(* Logix 5000 project; controller CarbonScout_MK6 vendor 1 type 14 code 154 rev 32.11; software revision 32.00; part 15 of 17 *)
(* tags used below, declared in another part *)
   CNT : DINT;
   DN_Cal : BOOL;   // Calculation Done Bit to proceed next step
   LocalSampleTank : DINT;
   LOnlineNumber : DINT;
   ONS : BOOL[32];
   SampleIndexNum : DINT;
   storage : BOOL;
   XRF_ReadyTimer : TIMER;
   CS_Alarms : P_Alarm[80];
   CS_DINTParams : DINT[100];
   CS_REALParams : REAL[80];   // CS REAL Parameters
   CS_Result : CS_Results;   // Sample Result Live Async
   CS_ResultsSync : CS_Results;
   CS_SampleSeq : DINT[129];
   CS_Seq : GEK_Sequence;
   CS_Tank : CS_TankParams[20];
   CS_Timer : TIMER[80];
   CS_Timer2 : TIMER[20];
   CS_XRF : XRF;
   CS_XRF_Elements : LinearModelXRF;   // Linear model 0 is inital factory model and 1 is trimming model
   CS_XRF_RawModel : REAL[4];
   N51 : DINT[5];   // From Client
   Oneshot : DINT;
   Oneshot2 : DINT;
   Oneshot3 : DINT;
   Reg_Model : REAL[4];   // Calculated model output and site model
   TankPointer : DINT;
   test : DINT;
   Valve_XV_15 : P_ValveSO;   // Bottme wash vavle
   Valve_XV_19 : P_ValveSO;   // Laser window
   Valve_XV_40 : P_ValveSO;   // XRF power on valve
   XRF_RAWDINT : DINT[100];
(* SeqProgram, continued *)

ROUTINE TankSelection   (* ladder *)
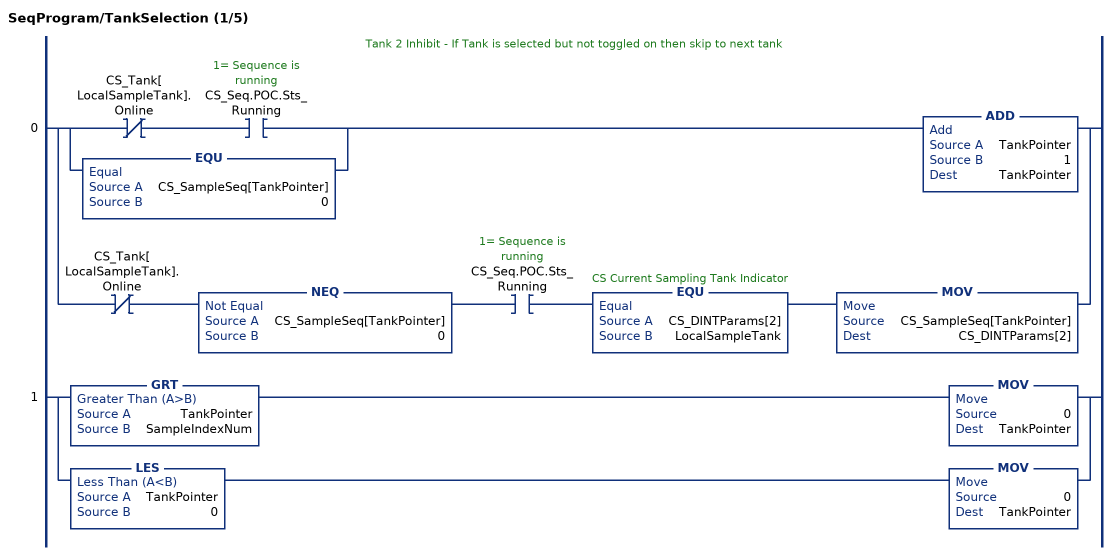
   // Tank 2 Inhibit - If Tank is selected but not toggled on then skip to next tank
   0: [[XIO(CS_Tank[LocalSampleTank].Online) XIC(CS_Seq.POC.Sts_Running) ,EQU(CS_SampleSeq[TankPointer],0) ] ADD(TankPointer,1,TankPointer) ,XIO(CS_Tank[LocalSampleTank].Online) NEQ(CS_SampleSeq[TankPointer],0) XIC(CS_Seq.POC.Sts_Running) EQU(CS_DINTParams[2],LocalSampleTank) MOV(CS_SampleSeq[TankPointer],CS_DINTParams[2]) ];
   1: [GRT(TankPointer,SampleIndexNum) MOV(0,TankPointer) ,LES(TankPointer,0) MOV(0,TankPointer) ];
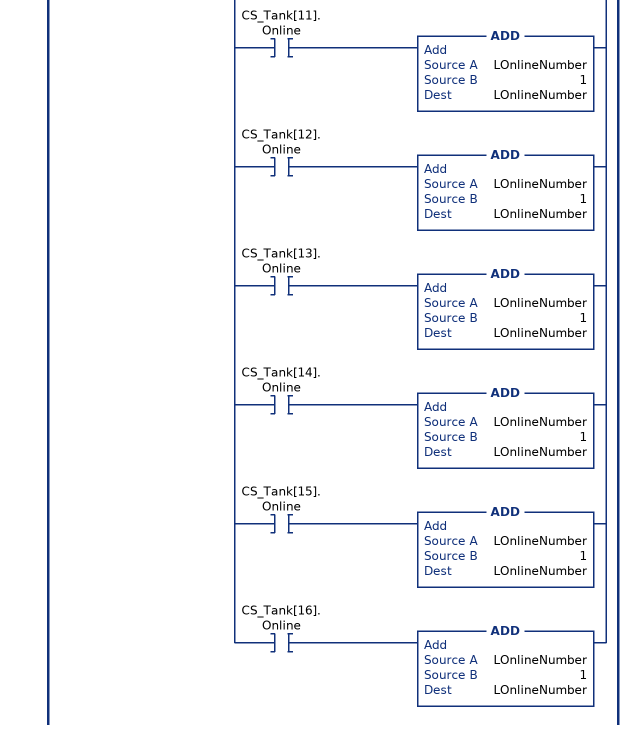
   2: CLR(LOnlineNumber)[XIC(CS_Tank[1].Online) ADD(LOnlineNumber,1,LOnlineNumber) ,XIC(CS_Tank[2].Online) ADD(LOnlineNumber,1,LOnlineNumber) ,XIC(CS_Tank[3].Online) ADD(LOnlineNumber,1,LOnlineNumber) ,XIC(CS_Tank[4].Online) ADD(LOnlineNumber,1,LOnlineNumber) ,XIC(CS_Tank[5].Online) ADD(LOnlineNumber,1,LOnlineNumber) ,XIC(CS_Tank[6].Online) ADD(LOnlineNumber,1,LOnlineNumber) ,XIC(CS_Tank[7].Online) ADD(LOnlineNumber,1,LOnlineNumber) ,XIC(CS_Tank[8].Online) ADD(LOnlineNumber,1,LOnlineNumber) ,XIC(CS_Tank[9].Online) ADD(LOnlineNumber,1,LOnlineNumber) ,XIC(CS_Tank[10].Online) ADD(LOnlineNumber,1,LOnlineNumber) ,XIC(CS_Tank[11].Online) ADD(LOnlineNumber,1,LOnlineNumber) ,XIC(CS_Tank[12].Online) ADD(LOnlineNumber,1,LOnlineNumber) ,XIC(CS_Tank[13].Online) ADD(LOnlineNumber,1,LOnlineNumber) ,XIC(CS_Tank[14].Online) ADD(LOnlineNumber,1,LOnlineNumber) ,XIC(CS_Tank[15].Online) ADD(LOnlineNumber,1,LOnlineNumber) ,XIC(CS_Tank[16].Online) ADD(LOnlineNumber,1,LOnlineNumber) ];
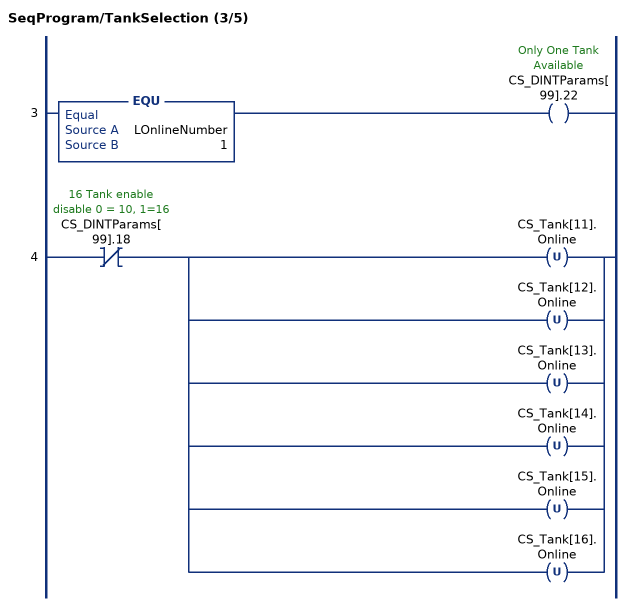
   3: EQU(LOnlineNumber,1)OTE(CS_DINTParams[99].22);
   4: XIO(CS_DINTParams[99].18)[OTU(CS_Tank[11].Online) ,OTU(CS_Tank[12].Online) ,OTU(CS_Tank[13].Online) ,OTU(CS_Tank[14].Online) ,OTU(CS_Tank[15].Online) ,OTU(CS_Tank[16].Online) ];
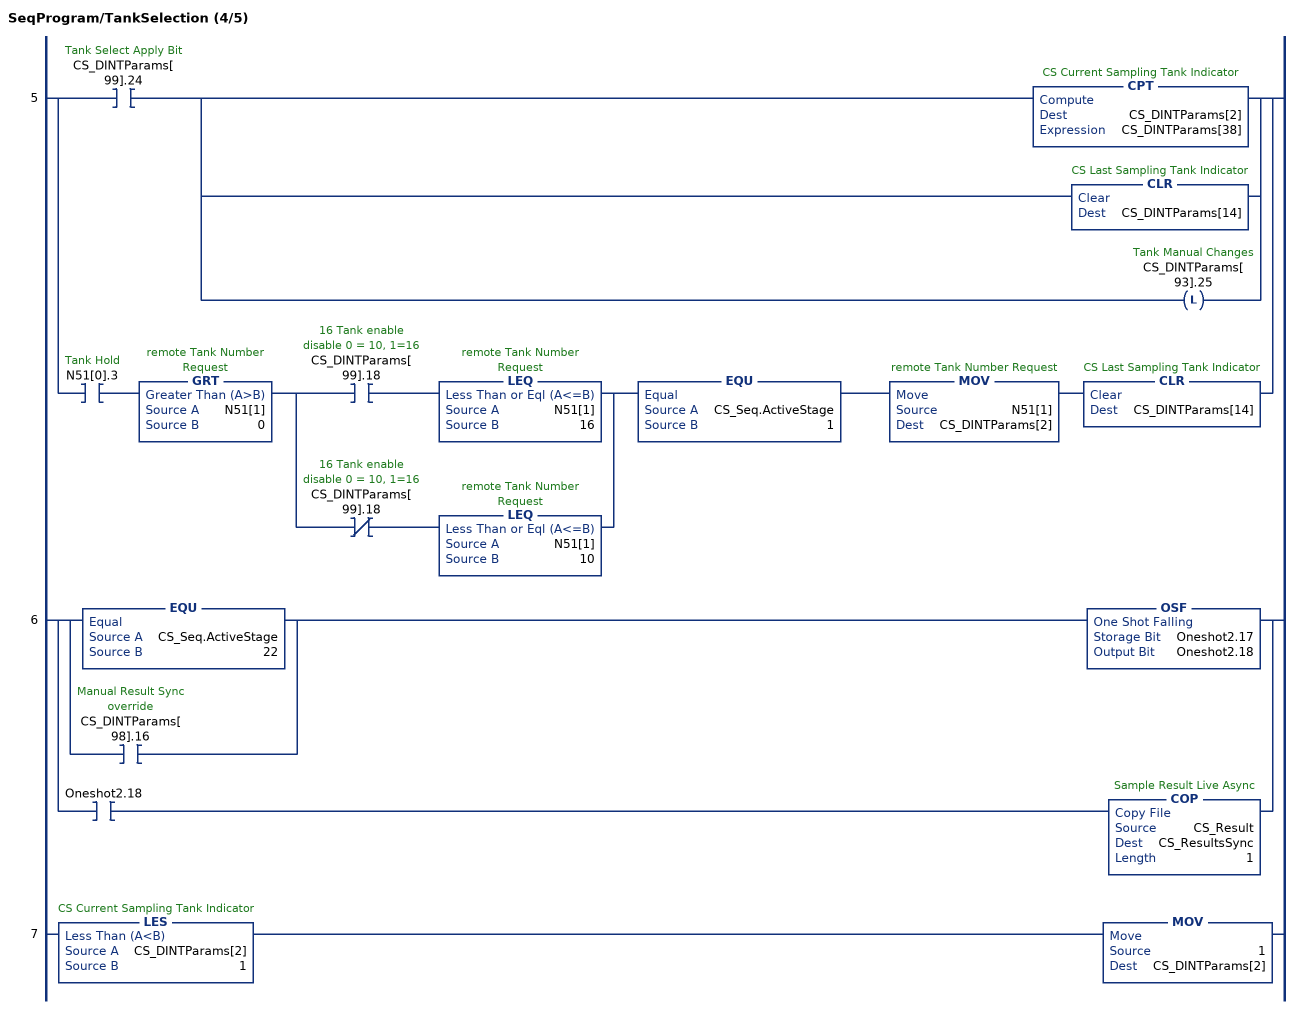
   5: [XIC(CS_DINTParams[99].24) [[CPT(CS_DINTParams[2],CS_DINTParams[38]) ,CLR(CS_DINTParams[14]) ] ,OTL(CS_DINTParams[93].25) ] ,XIC(N51[0].3) GRT(N51[1],0) [XIC(CS_DINTParams[99].18) LEQ(N51[1],16) ,XIO(CS_DINTParams[99].18) LEQ(N51[1],10) ] EQU(CS_Seq.ActiveStage,1) MOV(N51[1],CS_DINTParams[2]) CLR(CS_DINTParams[14]) ];
   6: [[EQU(CS_Seq.ActiveStage,22) ,XIC(CS_DINTParams[98].16) ] OSF(Oneshot2.17,Oneshot2.18) ,XIC(Oneshot2.18) COP(CS_Result,CS_ResultsSync,1) ];
   7: LES(CS_DINTParams[2],1)MOV(1,CS_DINTParams[2]);
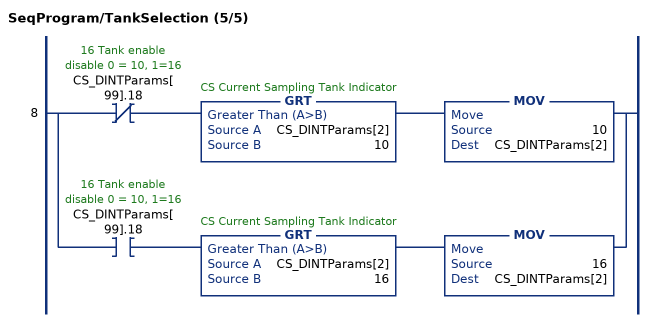
   8: [XIO(CS_DINTParams[99].18) GRT(CS_DINTParams[2],10) MOV(10,CS_DINTParams[2]) ,XIC(CS_DINTParams[99].18) GRT(CS_DINTParams[2],16) MOV(16,CS_DINTParams[2]) ];
END_ROUTINE

ROUTINE XRF   (* ladder *)
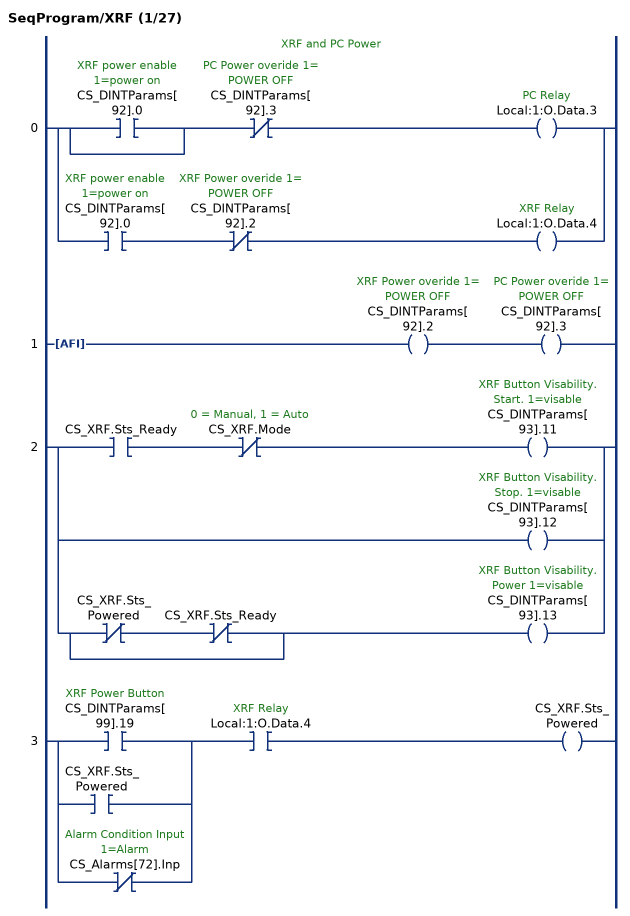
   // XRF and PC Power
   0: [[XIC(CS_DINTParams[92].0) ,] XIO(CS_DINTParams[92].3) OTE(Local:1:O.Data.3) ,XIC(CS_DINTParams[92].0) XIO(CS_DINTParams[92].2) OTE(Local:1:O.Data.4) ];
   1: AFI()OTE(CS_DINTParams[92].2)OTE(CS_DINTParams[92].3);
   2: [XIC(CS_XRF.Sts_Ready) XIO(CS_XRF.Mode) OTE(CS_DINTParams[93].11) ,OTE(CS_DINTParams[93].12) ,[XIO(CS_XRF.Sts_Powered) XIO(CS_XRF.Sts_Ready) ,] OTE(CS_DINTParams[93].13) ];
   3: [XIC(CS_DINTParams[99].19) ,XIC(CS_XRF.Sts_Powered) ,XIO(CS_Alarms[72].Inp) ]XIC(Local:1:O.Data.4)OTE(CS_XRF.Sts_Powered);
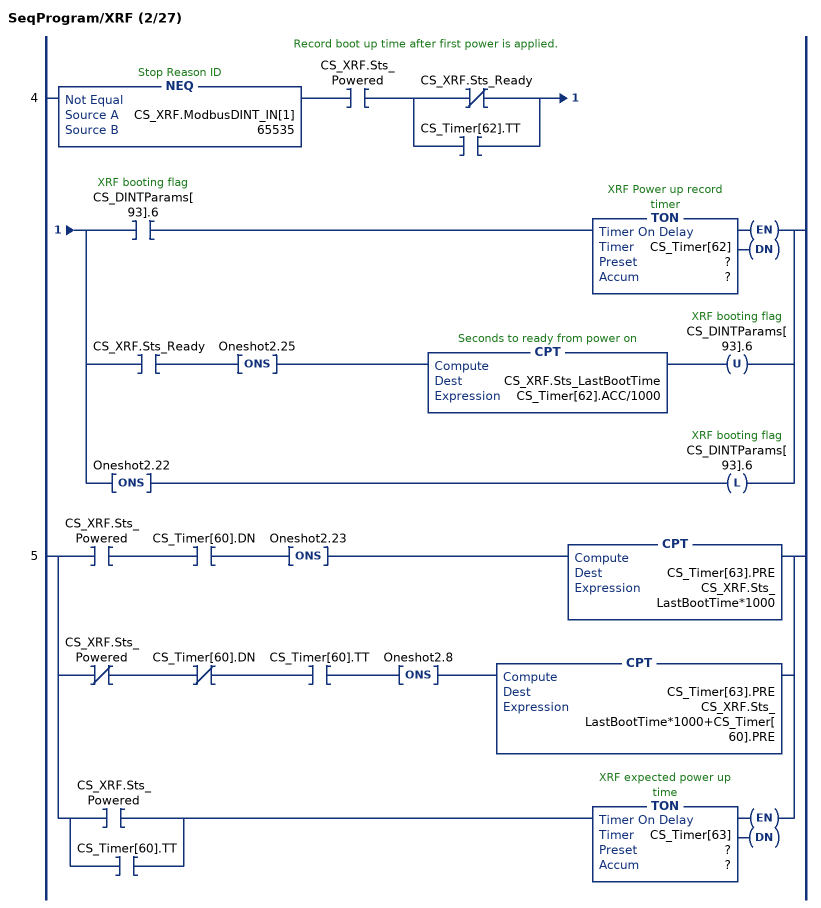
   // Record boot up time after first power is applied.
   4: NEQ(CS_XRF.ModbusDINT_IN[1],65535)XIC(CS_XRF.Sts_Powered)[XIO(CS_XRF.Sts_Ready) ,XIC(CS_Timer[62].TT) ][XIC(CS_DINTParams[93].6) TON(CS_Timer[62],?,?) ,XIC(CS_XRF.Sts_Ready) ONS(Oneshot2.25) CPT(CS_XRF.Sts_LastBootTime,CS_Timer[62].ACC/1000) OTU(CS_DINTParams[93].6) ,ONS(Oneshot2.22) OTL(CS_DINTParams[93].6) ];
   5: [XIC(CS_XRF.Sts_Powered) XIC(CS_Timer[60].DN) ONS(Oneshot2.23) CPT(CS_Timer[63].PRE,CS_XRF.Sts_LastBootTime*1000) ,XIO(CS_XRF.Sts_Powered) XIO(CS_Timer[60].DN) XIC(CS_Timer[60].TT) ONS(Oneshot2.8) CPT(CS_Timer[63].PRE,CS_XRF.Sts_LastBootTime*1000+CS_Timer[60].PRE) ,[XIC(CS_XRF.Sts_Powered) ,XIC(CS_Timer[60].TT) ] TON(CS_Timer[63],?,?) ];
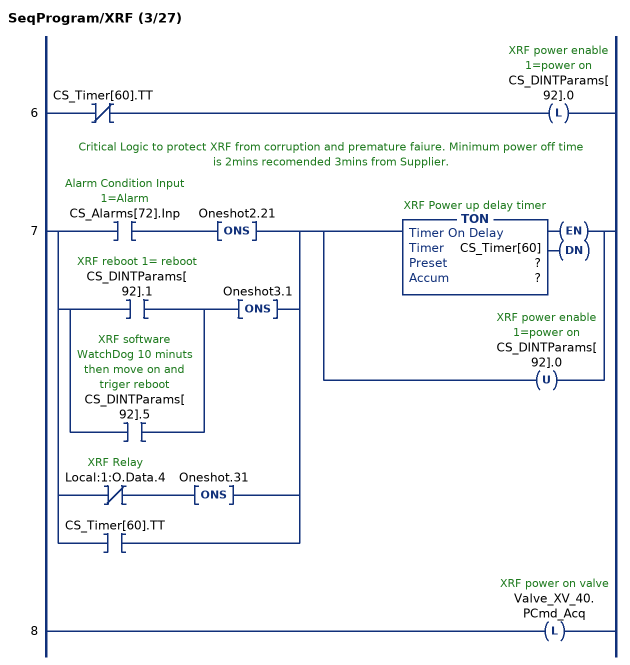
   6: XIO(CS_Timer[60].TT)OTL(CS_DINTParams[92].0);
   // Critical Logic to protect XRF from corruption and premature faiure. Minimum power off time is 2mins recomended 3mins from Supplier.
   7: [XIC(CS_Alarms[72].Inp) ONS(Oneshot2.21) ,[XIC(CS_DINTParams[92].1) ,XIC(CS_DINTParams[92].5) ] ONS(Oneshot3.1) ,XIO(Local:1:O.Data.4) ONS(Oneshot.31) ,XIC(CS_Timer[60].TT) ][TON(CS_Timer[60],?,?) ,OTU(CS_DINTParams[92].0) ];
   8: OTL(Valve_XV_40.PCmd_Acq);
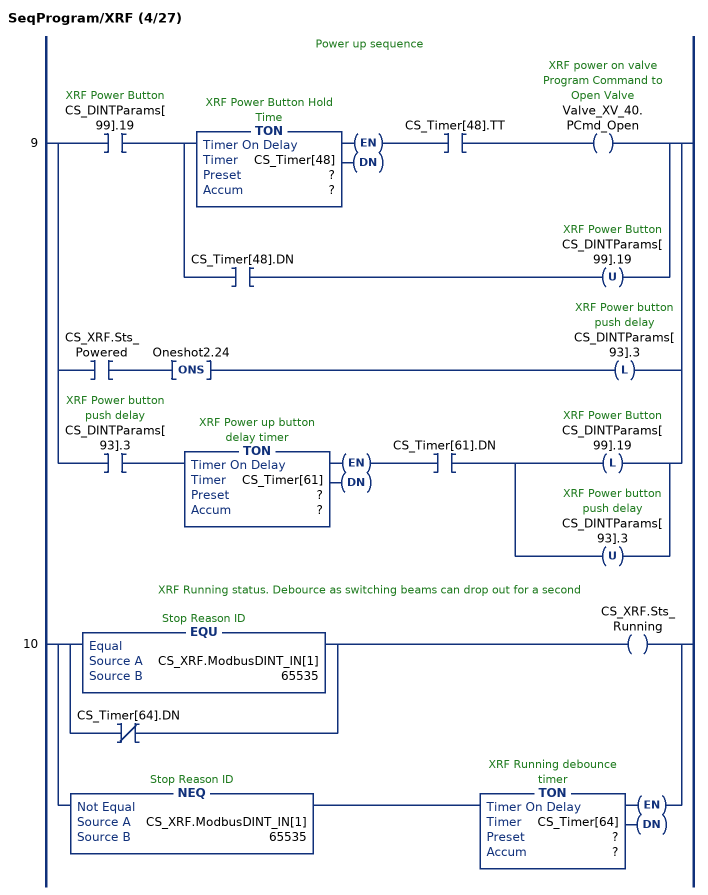
   // Power up sequence
   9: [XIC(CS_DINTParams[99].19) [TON(CS_Timer[48],?,?) XIC(CS_Timer[48].TT) OTE(Valve_XV_40.PCmd_Open) ,XIC(CS_Timer[48].DN) OTU(CS_DINTParams[99].19) ] ,XIC(CS_XRF.Sts_Powered) ONS(Oneshot2.24) OTL(CS_DINTParams[93].3) ,XIC(CS_DINTParams[93].3) TON(CS_Timer[61],?,?) XIC(CS_Timer[61].DN) [OTL(CS_DINTParams[99].19) ,OTU(CS_DINTParams[93].3) ] ];
   // XRF Running status. Debource as switching beams can drop out for a second
   10: [[EQU(CS_XRF.ModbusDINT_IN[1],65535) ,XIO(CS_Timer[64].DN) ] OTE(CS_XRF.Sts_Running) ,NEQ(CS_XRF.ModbusDINT_IN[1],65535) TON(CS_Timer[64],?,?) ];
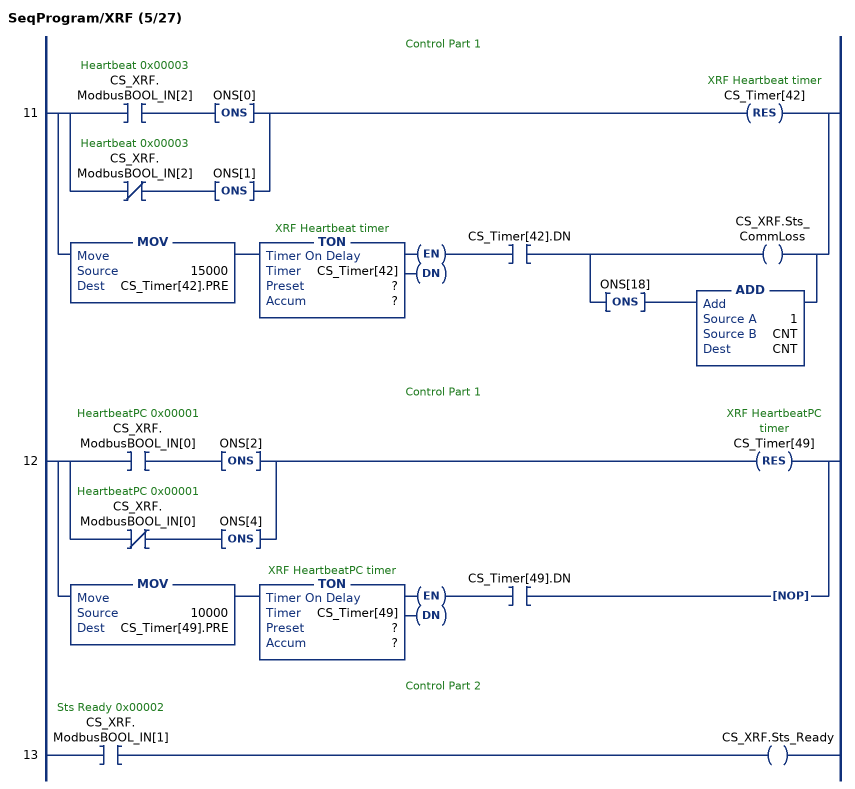
   // Control Part 1
   11: [[XIC(CS_XRF.ModbusBOOL_IN[2]) ONS(ONS[0]) ,XIO(CS_XRF.ModbusBOOL_IN[2]) ONS(ONS[1]) ] RES(CS_Timer[42]) ,MOV(15000,CS_Timer[42].PRE) TON(CS_Timer[42],?,?) XIC(CS_Timer[42].DN) [OTE(CS_XRF.Sts_CommLoss) ,ONS(ONS[18]) ADD(1,CNT,CNT) ] ];
   // Control Part 1
   12: [[XIC(CS_XRF.ModbusBOOL_IN[0]) ONS(ONS[2]) ,XIO(CS_XRF.ModbusBOOL_IN[0]) ONS(ONS[4]) ] RES(CS_Timer[49]) ,MOV(10000,CS_Timer[49].PRE) TON(CS_Timer[49],?,?) XIC(CS_Timer[49].DN) NOP() ];
   // Control Part 2
   13: XIC(CS_XRF.ModbusBOOL_IN[1])OTE(CS_XRF.Sts_Ready);
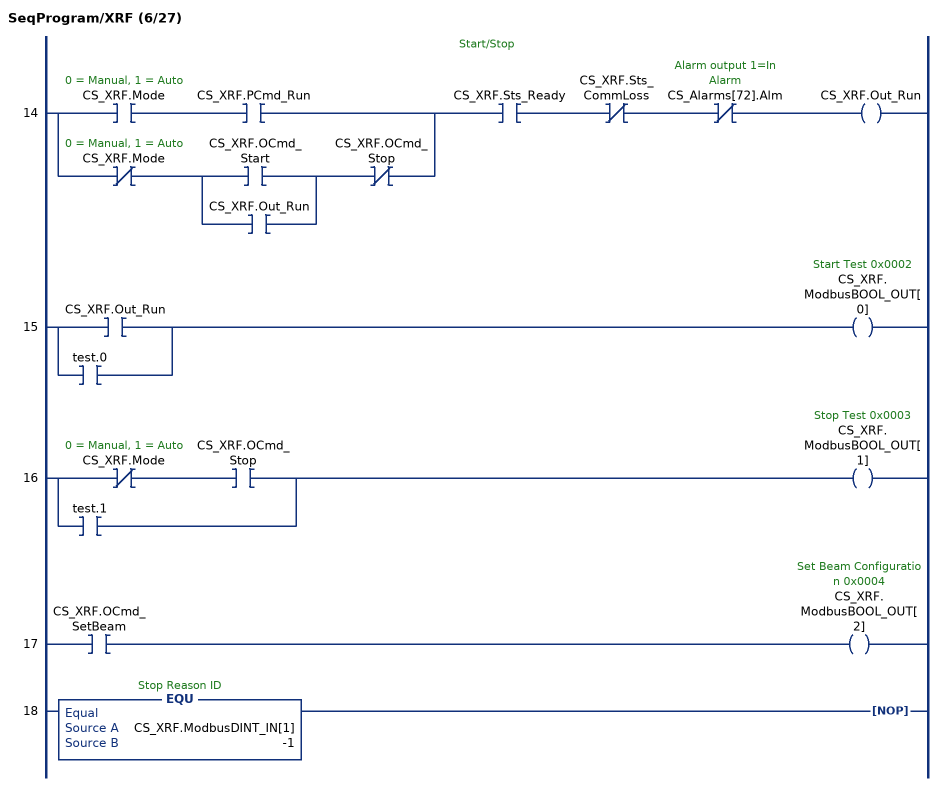
   // Start/Stop
   14: [XIC(CS_XRF.Mode) XIC(CS_XRF.PCmd_Run) ,XIO(CS_XRF.Mode) [XIC(CS_XRF.OCmd_Start) ,XIC(CS_XRF.Out_Run) ] XIO(CS_XRF.OCmd_Stop) ]XIC(CS_XRF.Sts_Ready)XIO(CS_XRF.Sts_CommLoss)XIO(CS_Alarms[72].Alm)OTE(CS_XRF.Out_Run);
   15: [XIC(CS_XRF.Out_Run) ,XIC(test.0) ]OTE(CS_XRF.ModbusBOOL_OUT[0]);
   16: [XIO(CS_XRF.Mode) XIC(CS_XRF.OCmd_Stop) ,XIC(test.1) ]OTE(CS_XRF.ModbusBOOL_OUT[1]);
   17: XIC(CS_XRF.OCmd_SetBeam)OTE(CS_XRF.ModbusBOOL_OUT[2]);
   18: EQU(CS_XRF.ModbusDINT_IN[1],-1)NOP();
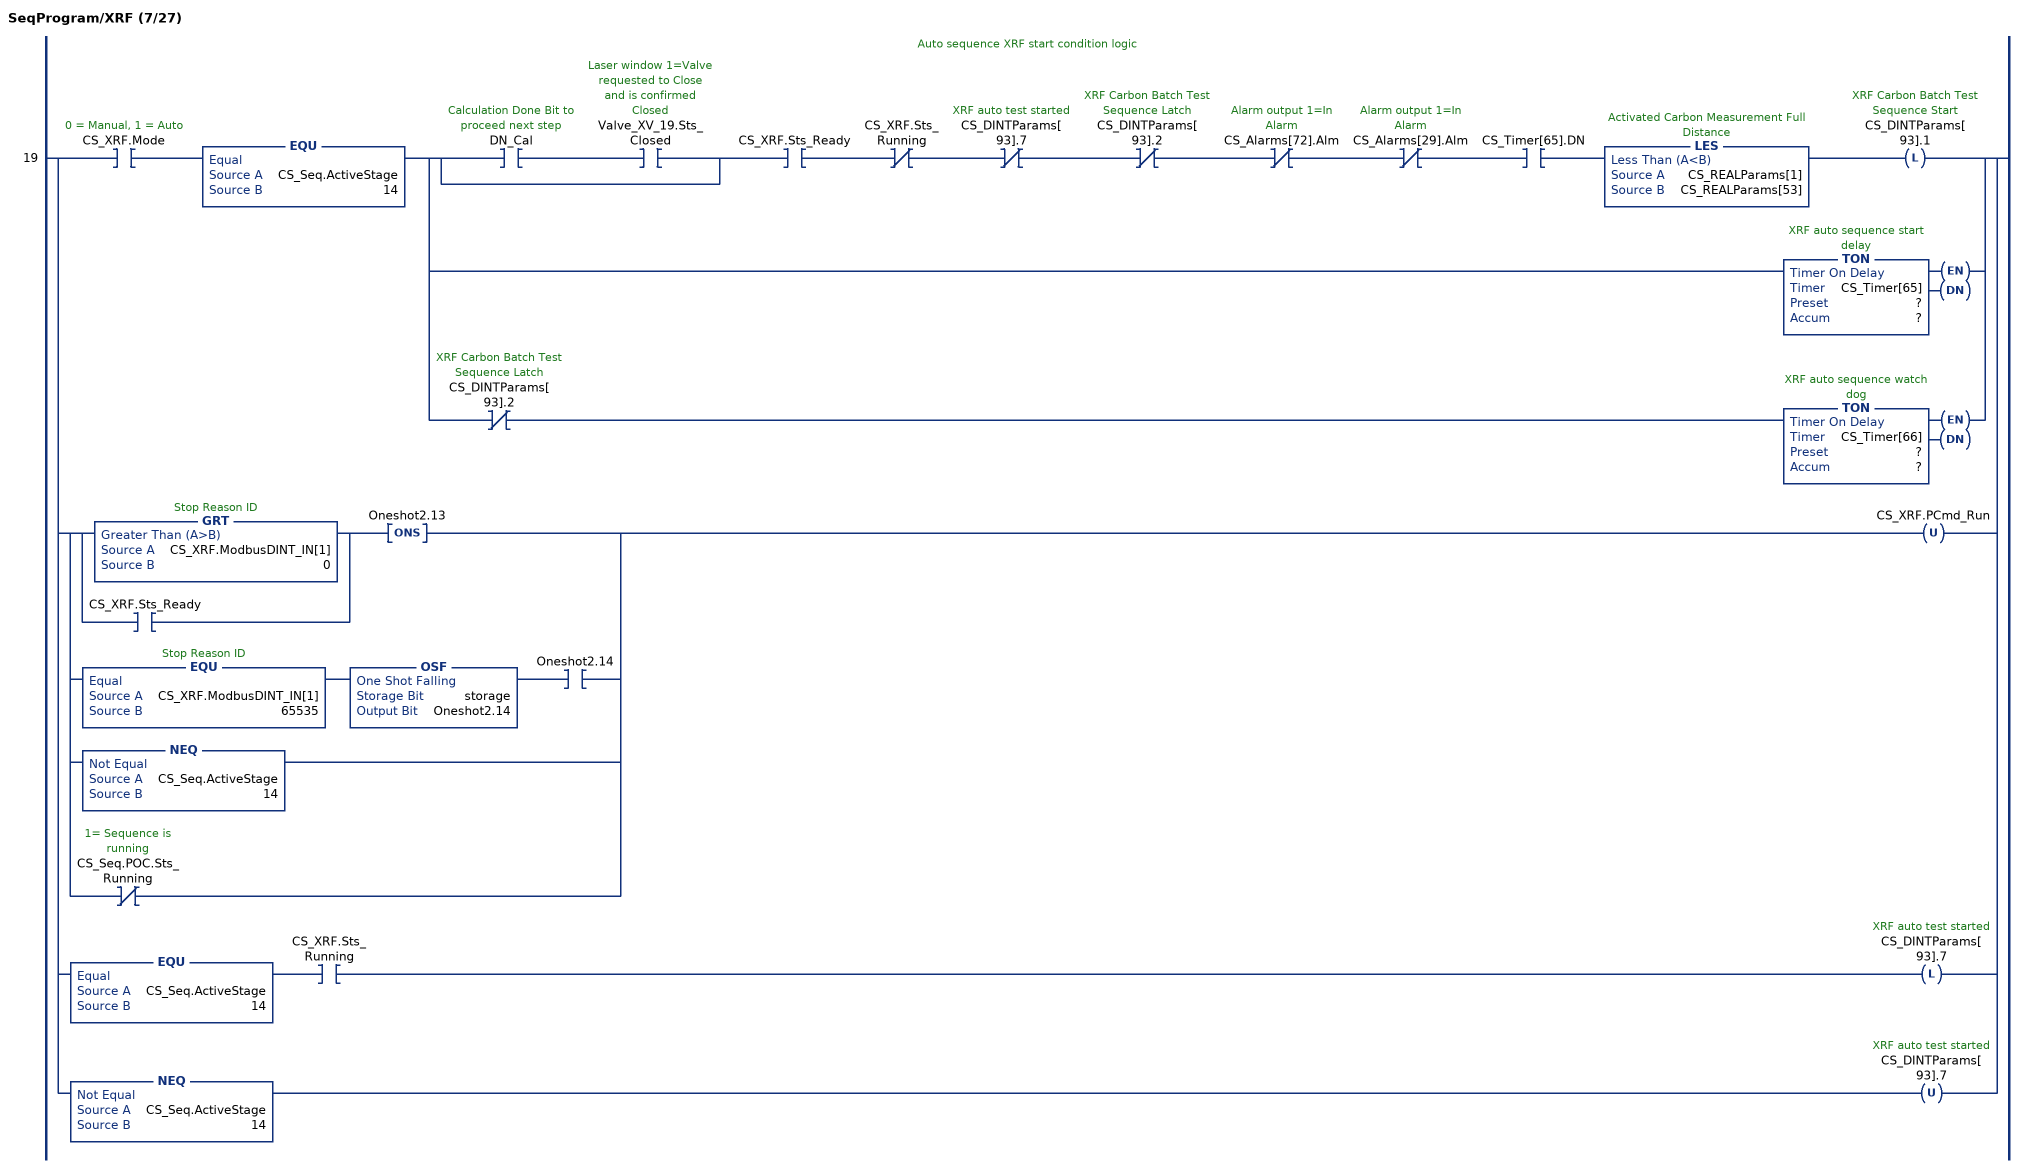
   // Auto sequence XRF start condition logic
   19: [XIC(CS_XRF.Mode) EQU(CS_Seq.ActiveStage,14) [[XIC(DN_Cal) XIC(Valve_XV_19.Sts_Closed) ,] XIC(CS_XRF.Sts_Ready) XIO(CS_XRF.Sts_Running) XIO(CS_DINTParams[93].7) XIO(CS_DINTParams[93].2) XIO(CS_Alarms[72].Alm) XIO(CS_Alarms[29].Alm) XIC(CS_Timer[65].DN) LES(CS_REALParams[1],CS_REALParams[53]) OTL(CS_DINTParams[93].1) ,[TON(CS_Timer[65],?,?) ,XIO(CS_DINTParams[93].2) TON(CS_Timer[66],?,?) ] ] ,[[GRT(CS_XRF.ModbusDINT_IN[1],0) ,XIC(CS_XRF.Sts_Ready) ] ONS(Oneshot2.13) ,EQU(CS_XRF.ModbusDINT_IN[1],65535) OSF(storage,Oneshot2.14) XIC(Oneshot2.14) ,NEQ(CS_Seq.ActiveStage,14) ,XIO(CS_Seq.POC.Sts_Running) ] OTU(CS_XRF.PCmd_Run) ,EQU(CS_Seq.ActiveStage,14) XIC(CS_XRF.Sts_Running) OTL(CS_DINTParams[93].7) ,NEQ(CS_Seq.ActiveStage,14) OTU(CS_DINTParams[93].7) ];
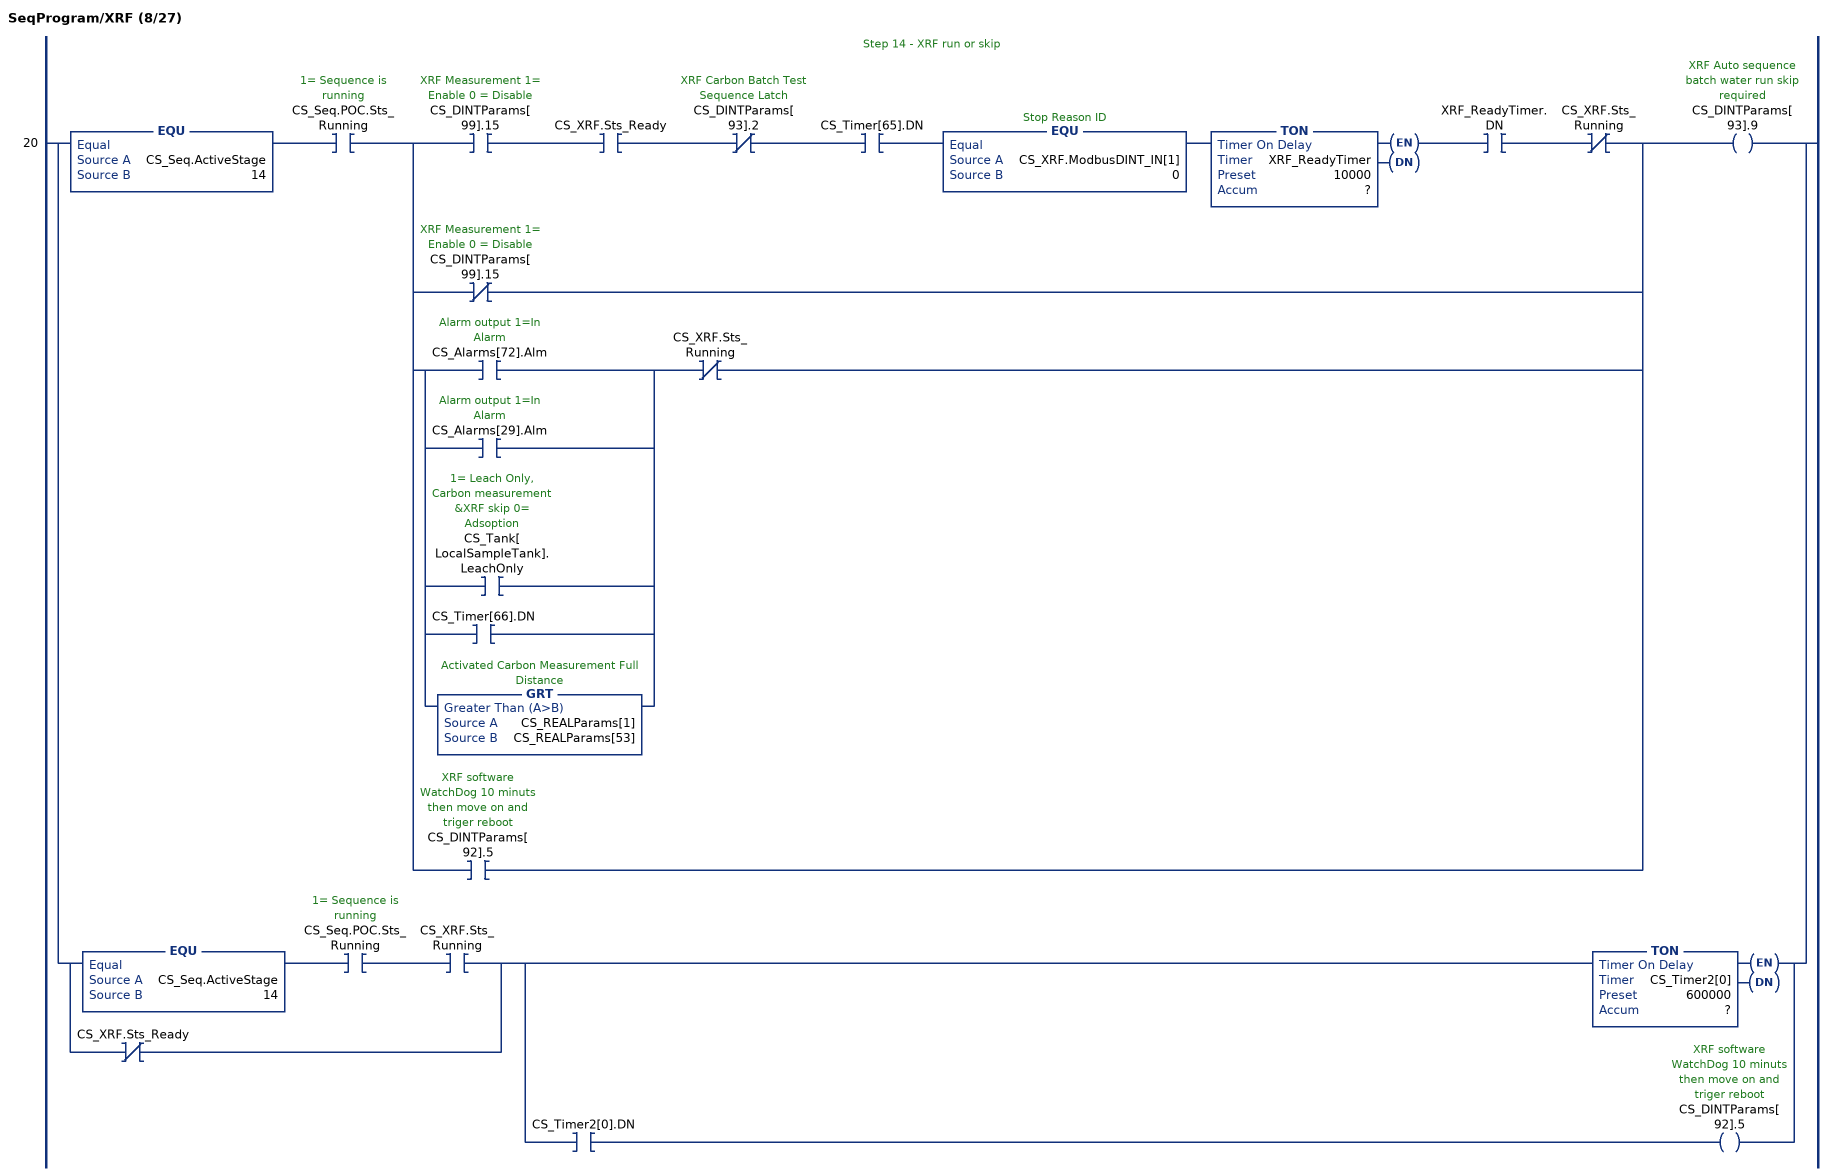
   // Step 14 - XRF run or skip
   20: [EQU(CS_Seq.ActiveStage,14) XIC(CS_Seq.POC.Sts_Running) [[XIC(CS_DINTParams[99].15) XIC(CS_XRF.Sts_Ready) XIO(CS_DINTParams[93].2) XIC(CS_Timer[65].DN) EQU(CS_XRF.ModbusDINT_IN[1],0) TON(XRF_ReadyTimer,?,?) XIC(XRF_ReadyTimer.DN) XIO(CS_XRF.Sts_Running) ,XIO(CS_DINTParams[99].15) ] ,[[XIC(CS_Alarms[72].Alm) ,XIC(CS_Alarms[29].Alm) ,XIC(CS_Tank[LocalSampleTank].LeachOnly) ,XIC(CS_Timer[66].DN) ,GRT(CS_REALParams[1],CS_REALParams[53]) ] XIO(CS_XRF.Sts_Running) ,XIC(CS_DINTParams[92].5) ] ] OTE(CS_DINTParams[93].9) ,[EQU(CS_Seq.ActiveStage,14) XIC(CS_Seq.POC.Sts_Running) XIC(CS_XRF.Sts_Running) ,XIO(CS_XRF.Sts_Ready) ] [TON(CS_Timer2[0],?,?) ,XIC(CS_Timer2[0].DN) OTE(CS_DINTParams[92].5) ] ];
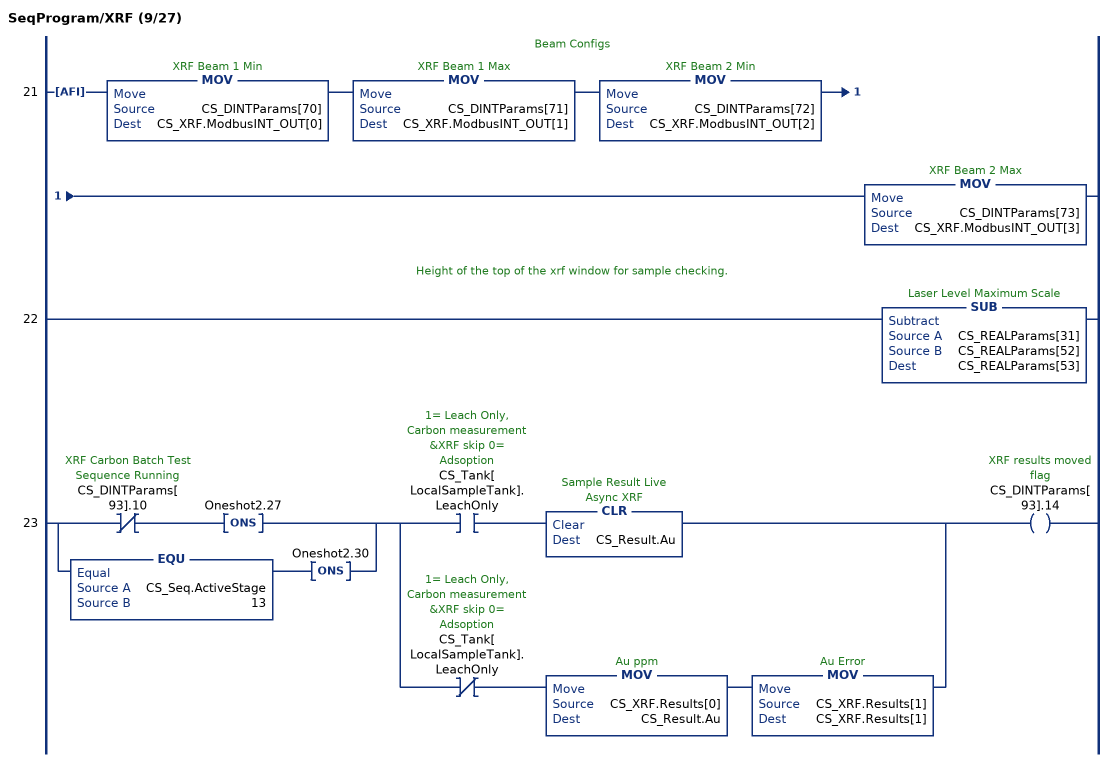
   // Beam Configs
   21: AFI()MOV(CS_DINTParams[70],CS_XRF.ModbusINT_OUT[0])MOV(CS_DINTParams[71],CS_XRF.ModbusINT_OUT[1])MOV(CS_DINTParams[72],CS_XRF.ModbusINT_OUT[2])MOV(CS_DINTParams[73],CS_XRF.ModbusINT_OUT[3]);
   // Height of the top of the xrf window for sample checking.
   22: SUB(CS_REALParams[31],CS_REALParams[52],CS_REALParams[53]);
   23: [XIO(CS_DINTParams[93].10) ONS(Oneshot2.27) ,EQU(CS_Seq.ActiveStage,13) ONS(Oneshot2.30) ][XIC(CS_Tank[LocalSampleTank].LeachOnly) CLR(CS_Result.Au) ,XIO(CS_Tank[LocalSampleTank].LeachOnly) MOV(CS_XRF.Results[0],CS_Result.Au) MOV(CS_XRF.Results[1],CS_XRF.Results[1]) ]OTE(CS_DINTParams[93].14);
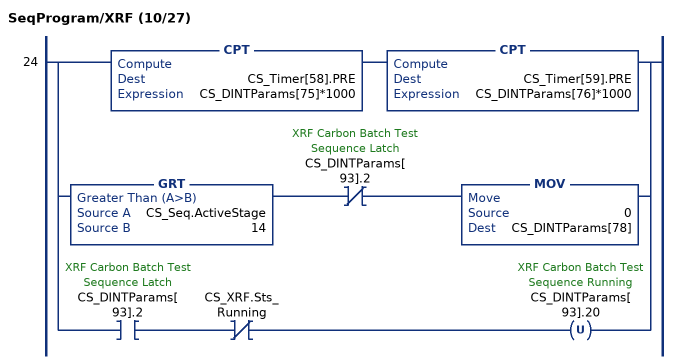
   24: [CPT(CS_Timer[58].PRE,CS_DINTParams[75]*1000) CPT(CS_Timer[59].PRE,CS_DINTParams[76]*1000) ,GRT(CS_Seq.ActiveStage,14) XIO(CS_DINTParams[93].2) MOV(0,CS_DINTParams[78]) ,XIC(CS_DINTParams[93].2) XIO(CS_XRF.Sts_Running) OTU(CS_DINTParams[93].20) ];
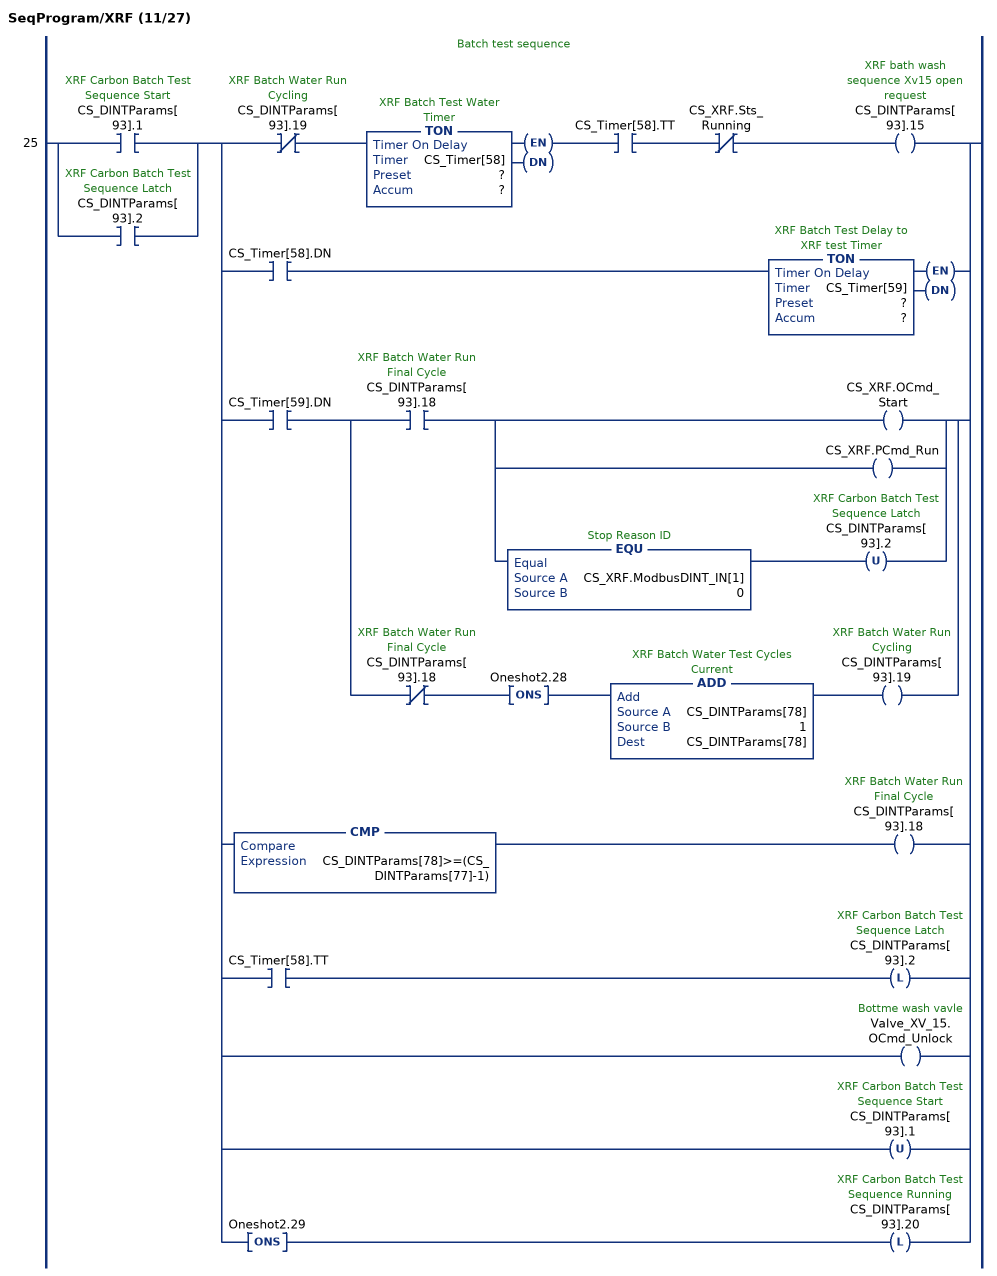
   // Batch test sequence
   25: [XIC(CS_DINTParams[93].1) ,XIC(CS_DINTParams[93].2) ][XIO(CS_DINTParams[93].19) TON(CS_Timer[58],?,?) XIC(CS_Timer[58].TT) XIO(CS_XRF.Sts_Running) OTE(CS_DINTParams[93].15) ,XIC(CS_Timer[58].DN) TON(CS_Timer[59],?,?) ,XIC(CS_Timer[59].DN) [XIC(CS_DINTParams[93].18) [[OTE(CS_XRF.OCmd_Start) ,OTE(CS_XRF.PCmd_Run) ] ,EQU(CS_XRF.ModbusDINT_IN[1],0) OTU(CS_DINTParams[93].2) ] ,XIO(CS_DINTParams[93].18) ONS(Oneshot2.28) ADD(CS_DINTParams[78],1,CS_DINTParams[78]) OTE(CS_DINTParams[93].19) ] ,CMP(CS_DINTParams[78]>=(CS_DINTParams[77]-1)) OTE(CS_DINTParams[93].18) ,XIC(CS_Timer[58].TT) OTL(CS_DINTParams[93].2) ,OTE(Valve_XV_15.OCmd_Unlock) ,OTU(CS_DINTParams[93].1) ,ONS(Oneshot2.29) OTL(CS_DINTParams[93].20) ];
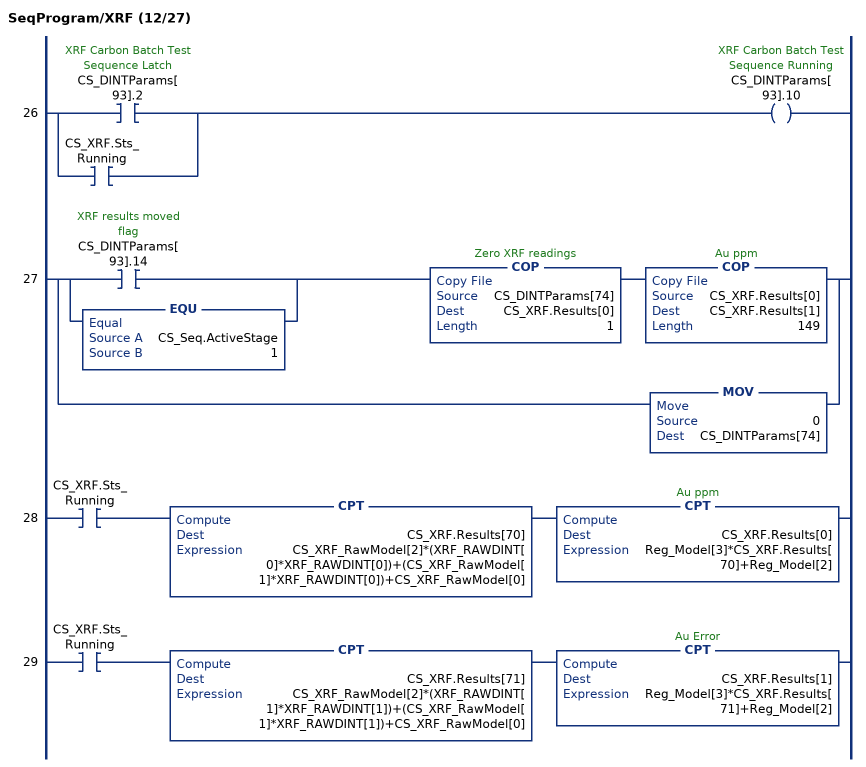
   26: [XIC(CS_DINTParams[93].2) ,XIC(CS_XRF.Sts_Running) ]OTE(CS_DINTParams[93].10);
   27: [[XIC(CS_DINTParams[93].14) ,EQU(CS_Seq.ActiveStage,1) ] COP(CS_DINTParams[74],CS_XRF.Results[0],1) COP(CS_XRF.Results[0],CS_XRF.Results[1],149) ,MOV(0,CS_DINTParams[74]) ];
   28: XIC(CS_XRF.Sts_Running)CPT(CS_XRF.Results[70],CS_XRF_RawModel[2]*(XRF_RAWDINT[0]*XRF_RAWDINT[0])+(CS_XRF_RawModel[1]*XRF_RAWDINT[0])+CS_XRF_RawModel[0])CPT(CS_XRF.Results[0],Reg_Model[3]*CS_XRF.Results[70]+Reg_Model[2]);
   29: XIC(CS_XRF.Sts_Running)CPT(CS_XRF.Results[71],CS_XRF_RawModel[2]*(XRF_RAWDINT[1]*XRF_RAWDINT[1])+(CS_XRF_RawModel[1]*XRF_RAWDINT[1])+CS_XRF_RawModel[0])CPT(CS_XRF.Results[1],Reg_Model[3]*CS_XRF.Results[71]+Reg_Model[2]);
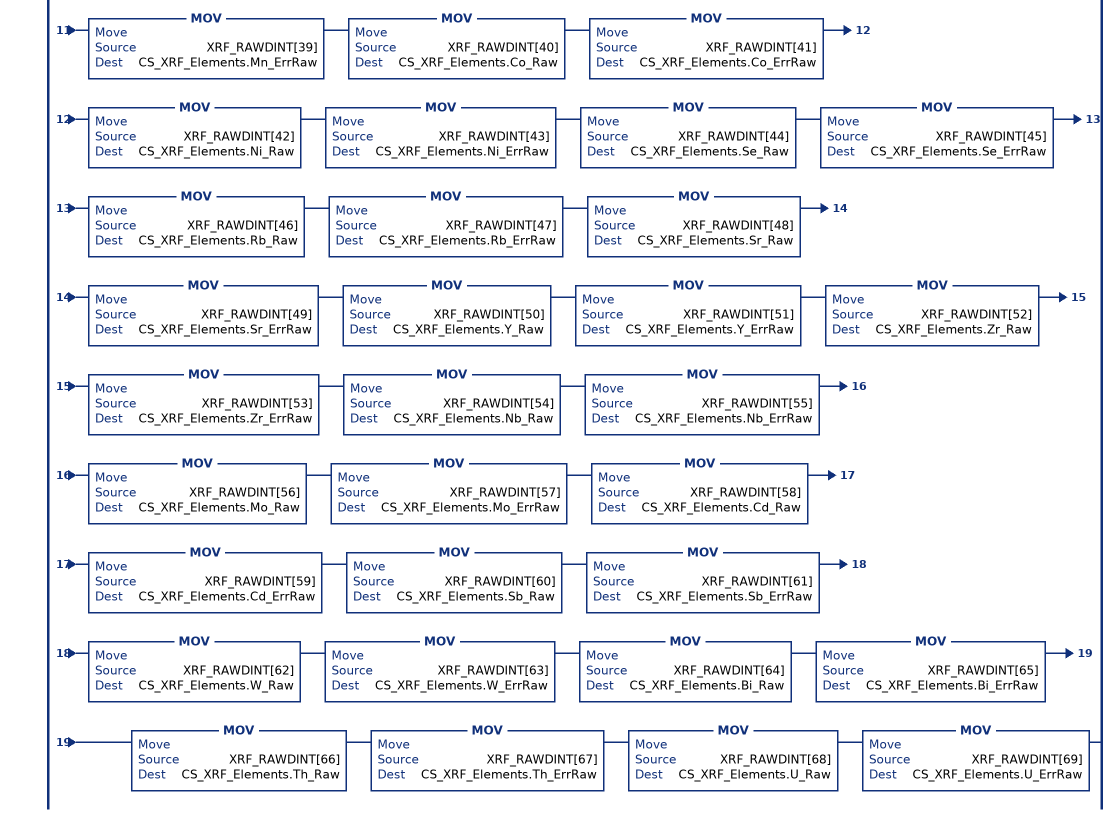
   30: MOV(XRF_RAWDINT[0],CS_XRF_Elements.Au_Raw)MOV(XRF_RAWDINT[1],CS_XRF_Elements.Au_ErrRaw)MOV(XRF_RAWDINT[2],CS_XRF_Elements.As_Raw)MOV(XRF_RAWDINT[3],CS_XRF_Elements.As_ErrRaw)MOV(XRF_RAWDINT[4],CS_XRF_Elements.Cu_Raw)MOV(XRF_RAWDINT[5],CS_XRF_Elements.Cu_ErrRaw)MOV(XRF_RAWDINT[6],CS_XRF_Elements.Fe_Raw)MOV(XRF_RAWDINT[7],CS_XRF_Elements.Fe_ErrRaw)MOV(XRF_RAWDINT[8],CS_XRF_Elements.Ag_Raw)MOV(XRF_RAWDINT[9],CS_XRF_Elements.Ag_ErrRaw)MOV(XRF_RAWDINT[10],CS_XRF_Elements.Hg_Raw)MOV(XRF_RAWDINT[11],CS_XRF_Elements.Hg_ErrRaw)MOV(XRF_RAWDINT[14],CS_XRF_Elements.Zn_Raw)MOV(XRF_RAWDINT[15],CS_XRF_Elements.Zn_ErrRaw)MOV(XRF_RAWDINT[16],CS_XRF_Elements.Sn_Raw)MOV(XRF_RAWDINT[17],CS_XRF_Elements.Sn_ErrRaw)MOV(XRF_RAWDINT[18],CS_XRF_Elements.Ca_Raw)MOV(XRF_RAWDINT[19],CS_XRF_Elements.Ca_ErrRaw)MOV(XRF_RAWDINT[20],CS_XRF_Elements.Mg_Raw)MOV(XRF_RAWDINT[21],CS_XRF_Elements.Mg_ErrRaw)MOV(XRF_RAWDINT[22],CS_XRF_Elements.Al_Raw)MOV(XRF_RAWDINT[23],CS_XRF_Elements.Al_ErrRaw)MOV(XRF_RAWDINT[24],CS_XRF_Elements.Si_Raw)MOV(XRF_RAWDINT[25],CS_XRF_Elements.Si_ErrRaw)MOV(XRF_RAWDINT[28],CS_XRF_Elements.S_Raw)MOV(XRF_RAWDINT[26],CS_XRF_Elements.Pb_Raw)MOV(XRF_RAWDINT[27],CS_XRF_Elements.Pb_ErrRaw)MOV(XRF_RAWDINT[29],CS_XRF_Elements.S_ErrRaw)MOV(XRF_RAWDINT[30],CS_XRF_Elements.K_Raw)MOV(XRF_RAWDINT[31],CS_XRF_Elements.K_ErrRaw)MOV(XRF_RAWDINT[32],CS_XRF_Elements.Ti_Raw)MOV(XRF_RAWDINT[33],CS_XRF_Elements.Ti_ErrRaw)MOV(XRF_RAWDINT[34],CS_XRF_Elements.V_Raw)MOV(XRF_RAWDINT[35],CS_XRF_Elements.V_ErrRaw)MOV(XRF_RAWDINT[36],CS_XRF_Elements.Cr_Raw)MOV(XRF_RAWDINT[37],CS_XRF_Elements.Cr_ErrRaw)MOV(XRF_RAWDINT[38],CS_XRF_Elements.Mn_Raw)MOV(XRF_RAWDINT[39],CS_XRF_Elements.Mn_ErrRaw)MOV(XRF_RAWDINT[40],CS_XRF_Elements.Co_Raw)MOV(XRF_RAWDINT[41],CS_XRF_Elements.Co_ErrRaw)MOV(XRF_RAWDINT[42],CS_XRF_Elements.Ni_Raw)MOV(XRF_RAWDINT[43],CS_XRF_Elements.Ni_ErrRaw)MOV(XRF_RAWDINT[44],CS_XRF_Elements.Se_Raw)MOV(XRF_RAWDINT[45],CS_XRF_Elements.Se_ErrRaw)MOV(XRF_RAWDINT[46],CS_XRF_Elements.Rb_Raw)MOV(XRF_RAWDINT[47],CS_XRF_Elements.Rb_ErrRaw)MOV(XRF_RAWDINT[48],CS_XRF_Elements.Sr_Raw)MOV(XRF_RAWDINT[49],CS_XRF_Elements.Sr_ErrRaw)MOV(XRF_RAWDINT[50],CS_XRF_Elements.Y_Raw)MOV(XRF_RAWDINT[51],CS_XRF_Elements.Y_ErrRaw)MOV(XRF_RAWDINT[52],CS_XRF_Elements.Zr_Raw)MOV(XRF_RAWDINT[53],CS_XRF_Elements.Zr_ErrRaw)MOV(XRF_RAWDINT[54],CS_XRF_Elements.Nb_Raw)MOV(XRF_RAWDINT[55],CS_XRF_Elements.Nb_ErrRaw)MOV(XRF_RAWDINT[56],CS_XRF_Elements.Mo_Raw)MOV(XRF_RAWDINT[57],CS_XRF_Elements.Mo_ErrRaw)MOV(XRF_RAWDINT[58],CS_XRF_Elements.Cd_Raw)MOV(XRF_RAWDINT[59],CS_XRF_Elements.Cd_ErrRaw)MOV(XRF_RAWDINT[60],CS_XRF_Elements.Sb_Raw)MOV(XRF_RAWDINT[61],CS_XRF_Elements.Sb_ErrRaw)MOV(XRF_RAWDINT[62],CS_XRF_Elements.W_Raw)MOV(XRF_RAWDINT[63],CS_XRF_Elements.W_ErrRaw)MOV(XRF_RAWDINT[64],CS_XRF_Elements.Bi_Raw)MOV(XRF_RAWDINT[65],CS_XRF_Elements.Bi_ErrRaw)MOV(XRF_RAWDINT[66],CS_XRF_Elements.Th_Raw)MOV(XRF_RAWDINT[67],CS_XRF_Elements.Th_ErrRaw)MOV(XRF_RAWDINT[68],CS_XRF_Elements.U_Raw)MOV(XRF_RAWDINT[69],CS_XRF_Elements.U_ErrRaw);
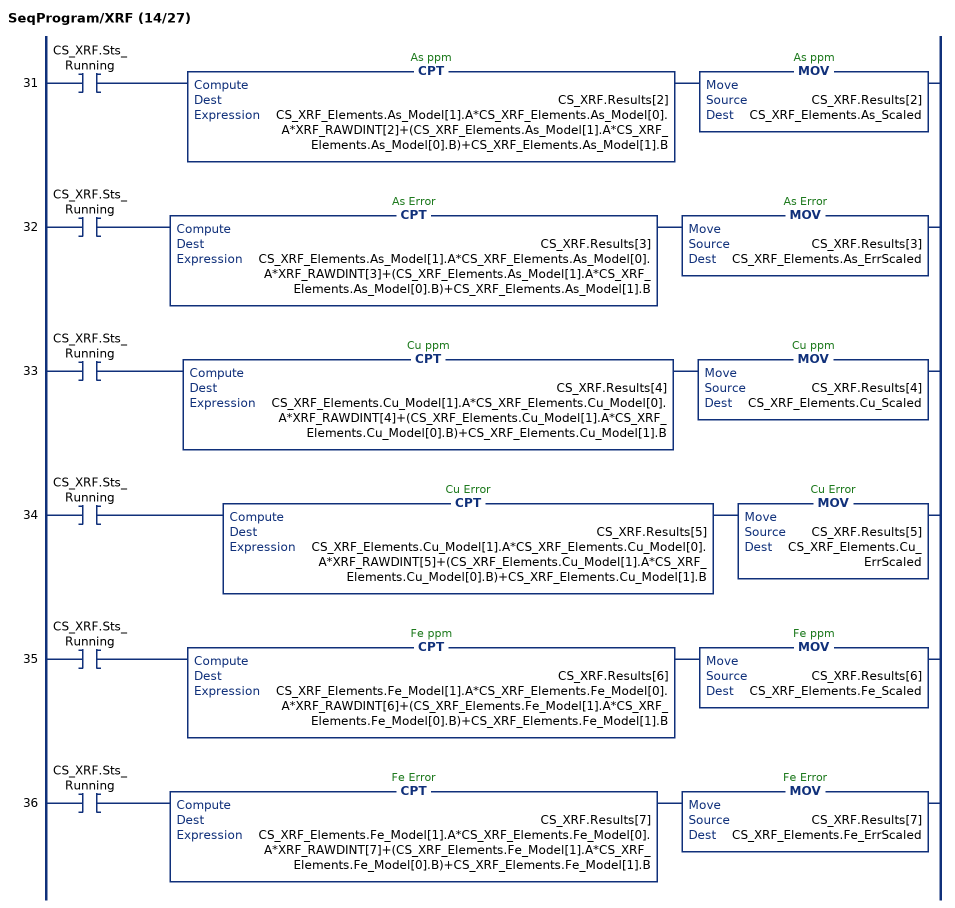
   31: XIC(CS_XRF.Sts_Running)CPT(CS_XRF.Results[2],CS_XRF_Elements.As_Model[1].A*CS_XRF_Elements.As_Model[0].A*XRF_RAWDINT[2]+(CS_XRF_Elements.As_Model[1].A*CS_XRF_Elements.As_Model[0].B)+CS_XRF_Elements.As_Model[1].B)MOV(CS_XRF.Results[2],CS_XRF_Elements.As_Scaled);
   32: XIC(CS_XRF.Sts_Running)CPT(CS_XRF.Results[3],CS_XRF_Elements.As_Model[1].A*CS_XRF_Elements.As_Model[0].A*XRF_RAWDINT[3]+(CS_XRF_Elements.As_Model[1].A*CS_XRF_Elements.As_Model[0].B)+CS_XRF_Elements.As_Model[1].B)MOV(CS_XRF.Results[3],CS_XRF_Elements.As_ErrScaled);
   33: XIC(CS_XRF.Sts_Running)CPT(CS_XRF.Results[4],CS_XRF_Elements.Cu_Model[1].A*CS_XRF_Elements.Cu_Model[0].A*XRF_RAWDINT[4]+(CS_XRF_Elements.Cu_Model[1].A*CS_XRF_Elements.Cu_Model[0].B)+CS_XRF_Elements.Cu_Model[1].B)MOV(CS_XRF.Results[4],CS_XRF_Elements.Cu_Scaled);
   34: XIC(CS_XRF.Sts_Running)CPT(CS_XRF.Results[5],CS_XRF_Elements.Cu_Model[1].A*CS_XRF_Elements.Cu_Model[0].A*XRF_RAWDINT[5]+(CS_XRF_Elements.Cu_Model[1].A*CS_XRF_Elements.Cu_Model[0].B)+CS_XRF_Elements.Cu_Model[1].B)MOV(CS_XRF.Results[5],CS_XRF_Elements.Cu_ErrScaled);
   35: XIC(CS_XRF.Sts_Running)CPT(CS_XRF.Results[6],CS_XRF_Elements.Fe_Model[1].A*CS_XRF_Elements.Fe_Model[0].A*XRF_RAWDINT[6]+(CS_XRF_Elements.Fe_Model[1].A*CS_XRF_Elements.Fe_Model[0].B)+CS_XRF_Elements.Fe_Model[1].B)MOV(CS_XRF.Results[6],CS_XRF_Elements.Fe_Scaled);
   36: XIC(CS_XRF.Sts_Running)CPT(CS_XRF.Results[7],CS_XRF_Elements.Fe_Model[1].A*CS_XRF_Elements.Fe_Model[0].A*XRF_RAWDINT[7]+(CS_XRF_Elements.Fe_Model[1].A*CS_XRF_Elements.Fe_Model[0].B)+CS_XRF_Elements.Fe_Model[1].B)MOV(CS_XRF.Results[7],CS_XRF_Elements.Fe_ErrScaled);
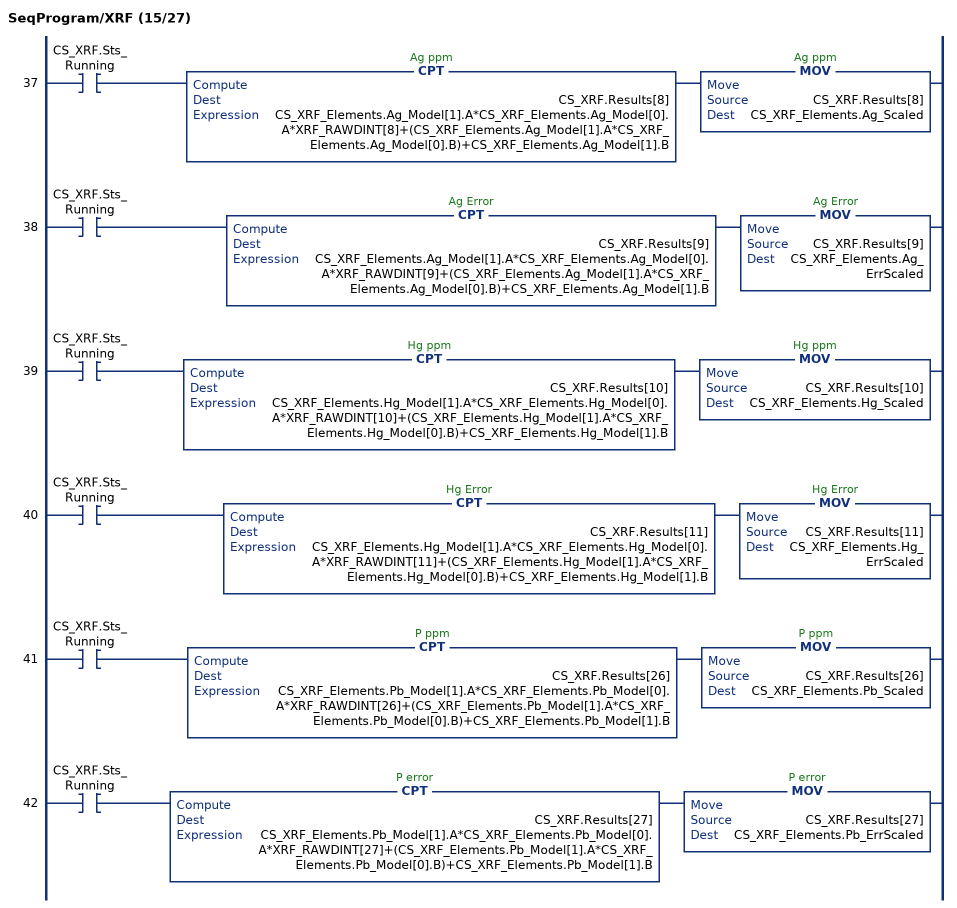
   37: XIC(CS_XRF.Sts_Running)CPT(CS_XRF.Results[8],CS_XRF_Elements.Ag_Model[1].A*CS_XRF_Elements.Ag_Model[0].A*XRF_RAWDINT[8]+(CS_XRF_Elements.Ag_Model[1].A*CS_XRF_Elements.Ag_Model[0].B)+CS_XRF_Elements.Ag_Model[1].B)MOV(CS_XRF.Results[8],CS_XRF_Elements.Ag_Scaled);
   38: XIC(CS_XRF.Sts_Running)CPT(CS_XRF.Results[9],CS_XRF_Elements.Ag_Model[1].A*CS_XRF_Elements.Ag_Model[0].A*XRF_RAWDINT[9]+(CS_XRF_Elements.Ag_Model[1].A*CS_XRF_Elements.Ag_Model[0].B)+CS_XRF_Elements.Ag_Model[1].B)MOV(CS_XRF.Results[9],CS_XRF_Elements.Ag_ErrScaled);
   39: XIC(CS_XRF.Sts_Running)CPT(CS_XRF.Results[10],CS_XRF_Elements.Hg_Model[1].A*CS_XRF_Elements.Hg_Model[0].A*XRF_RAWDINT[10]+(CS_XRF_Elements.Hg_Model[1].A*CS_XRF_Elements.Hg_Model[0].B)+CS_XRF_Elements.Hg_Model[1].B)MOV(CS_XRF.Results[10],CS_XRF_Elements.Hg_Scaled);
   40: XIC(CS_XRF.Sts_Running)CPT(CS_XRF.Results[11],CS_XRF_Elements.Hg_Model[1].A*CS_XRF_Elements.Hg_Model[0].A*XRF_RAWDINT[11]+(CS_XRF_Elements.Hg_Model[1].A*CS_XRF_Elements.Hg_Model[0].B)+CS_XRF_Elements.Hg_Model[1].B)MOV(CS_XRF.Results[11],CS_XRF_Elements.Hg_ErrScaled);
   41: XIC(CS_XRF.Sts_Running)CPT(CS_XRF.Results[26],CS_XRF_Elements.Pb_Model[1].A*CS_XRF_Elements.Pb_Model[0].A*XRF_RAWDINT[26]+(CS_XRF_Elements.Pb_Model[1].A*CS_XRF_Elements.Pb_Model[0].B)+CS_XRF_Elements.Pb_Model[1].B)MOV(CS_XRF.Results[26],CS_XRF_Elements.Pb_Scaled);
   42: XIC(CS_XRF.Sts_Running)CPT(CS_XRF.Results[27],CS_XRF_Elements.Pb_Model[1].A*CS_XRF_Elements.Pb_Model[0].A*XRF_RAWDINT[27]+(CS_XRF_Elements.Pb_Model[1].A*CS_XRF_Elements.Pb_Model[0].B)+CS_XRF_Elements.Pb_Model[1].B)MOV(CS_XRF.Results[27],CS_XRF_Elements.Pb_ErrScaled);
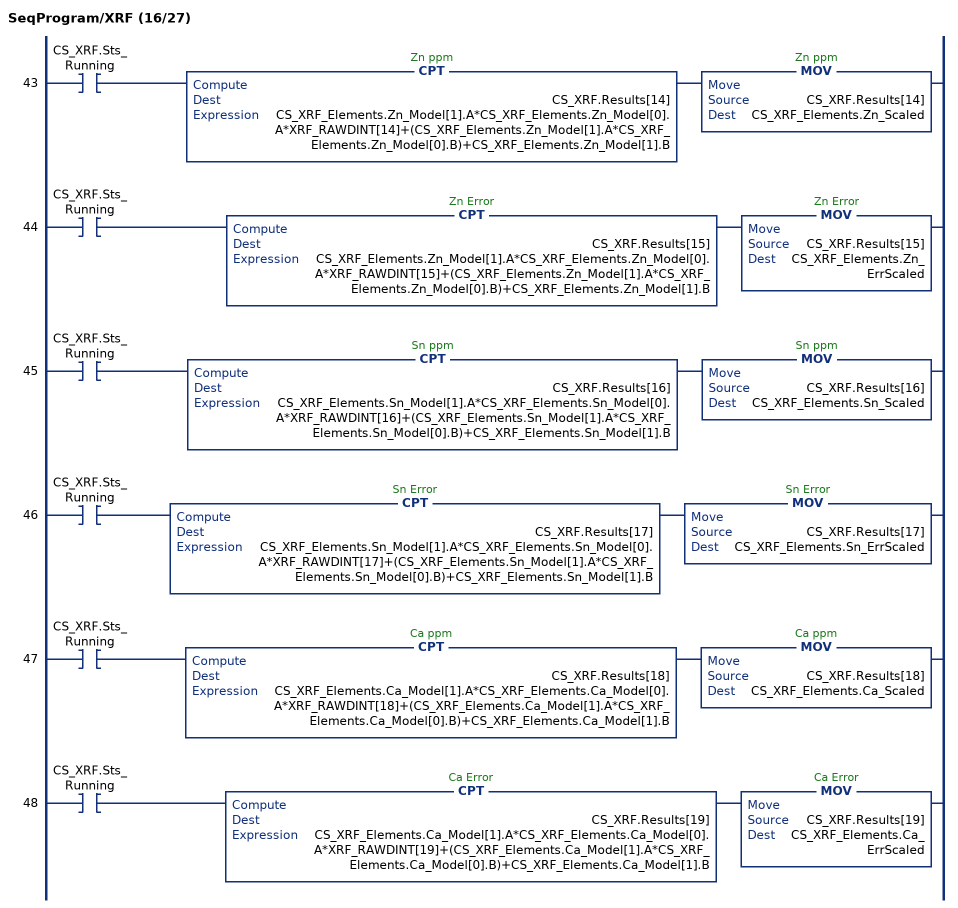
   43: XIC(CS_XRF.Sts_Running)CPT(CS_XRF.Results[14],CS_XRF_Elements.Zn_Model[1].A*CS_XRF_Elements.Zn_Model[0].A*XRF_RAWDINT[14]+(CS_XRF_Elements.Zn_Model[1].A*CS_XRF_Elements.Zn_Model[0].B)+CS_XRF_Elements.Zn_Model[1].B)MOV(CS_XRF.Results[14],CS_XRF_Elements.Zn_Scaled);
   44: XIC(CS_XRF.Sts_Running)CPT(CS_XRF.Results[15],CS_XRF_Elements.Zn_Model[1].A*CS_XRF_Elements.Zn_Model[0].A*XRF_RAWDINT[15]+(CS_XRF_Elements.Zn_Model[1].A*CS_XRF_Elements.Zn_Model[0].B)+CS_XRF_Elements.Zn_Model[1].B)MOV(CS_XRF.Results[15],CS_XRF_Elements.Zn_ErrScaled);
   45: XIC(CS_XRF.Sts_Running)CPT(CS_XRF.Results[16],CS_XRF_Elements.Sn_Model[1].A*CS_XRF_Elements.Sn_Model[0].A*XRF_RAWDINT[16]+(CS_XRF_Elements.Sn_Model[1].A*CS_XRF_Elements.Sn_Model[0].B)+CS_XRF_Elements.Sn_Model[1].B)MOV(CS_XRF.Results[16],CS_XRF_Elements.Sn_Scaled);
   46: XIC(CS_XRF.Sts_Running)CPT(CS_XRF.Results[17],CS_XRF_Elements.Sn_Model[1].A*CS_XRF_Elements.Sn_Model[0].A*XRF_RAWDINT[17]+(CS_XRF_Elements.Sn_Model[1].A*CS_XRF_Elements.Sn_Model[0].B)+CS_XRF_Elements.Sn_Model[1].B)MOV(CS_XRF.Results[17],CS_XRF_Elements.Sn_ErrScaled);
   47: XIC(CS_XRF.Sts_Running)CPT(CS_XRF.Results[18],CS_XRF_Elements.Ca_Model[1].A*CS_XRF_Elements.Ca_Model[0].A*XRF_RAWDINT[18]+(CS_XRF_Elements.Ca_Model[1].A*CS_XRF_Elements.Ca_Model[0].B)+CS_XRF_Elements.Ca_Model[1].B)MOV(CS_XRF.Results[18],CS_XRF_Elements.Ca_Scaled);
   48: XIC(CS_XRF.Sts_Running)CPT(CS_XRF.Results[19],CS_XRF_Elements.Ca_Model[1].A*CS_XRF_Elements.Ca_Model[0].A*XRF_RAWDINT[19]+(CS_XRF_Elements.Ca_Model[1].A*CS_XRF_Elements.Ca_Model[0].B)+CS_XRF_Elements.Ca_Model[1].B)MOV(CS_XRF.Results[19],CS_XRF_Elements.Ca_ErrScaled);
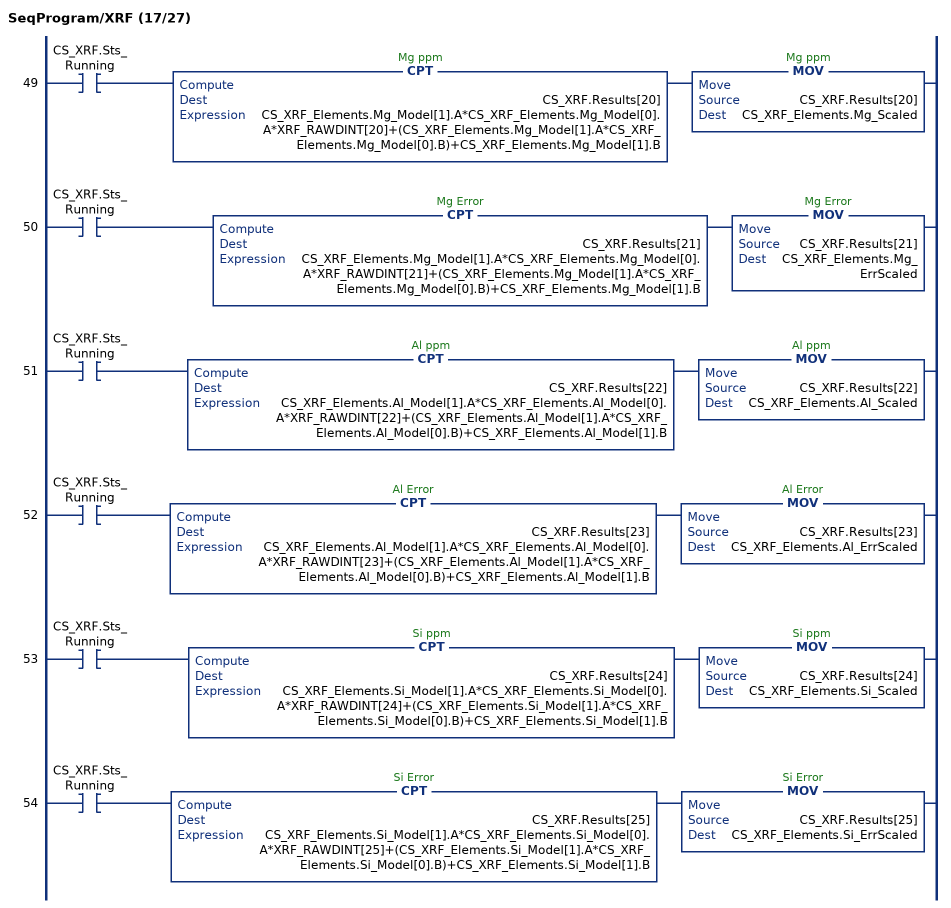
   49: XIC(CS_XRF.Sts_Running)CPT(CS_XRF.Results[20],CS_XRF_Elements.Mg_Model[1].A*CS_XRF_Elements.Mg_Model[0].A*XRF_RAWDINT[20]+(CS_XRF_Elements.Mg_Model[1].A*CS_XRF_Elements.Mg_Model[0].B)+CS_XRF_Elements.Mg_Model[1].B)MOV(CS_XRF.Results[20],CS_XRF_Elements.Mg_Scaled);
   50: XIC(CS_XRF.Sts_Running)CPT(CS_XRF.Results[21],CS_XRF_Elements.Mg_Model[1].A*CS_XRF_Elements.Mg_Model[0].A*XRF_RAWDINT[21]+(CS_XRF_Elements.Mg_Model[1].A*CS_XRF_Elements.Mg_Model[0].B)+CS_XRF_Elements.Mg_Model[1].B)MOV(CS_XRF.Results[21],CS_XRF_Elements.Mg_ErrScaled);
   51: XIC(CS_XRF.Sts_Running)CPT(CS_XRF.Results[22],CS_XRF_Elements.Al_Model[1].A*CS_XRF_Elements.Al_Model[0].A*XRF_RAWDINT[22]+(CS_XRF_Elements.Al_Model[1].A*CS_XRF_Elements.Al_Model[0].B)+CS_XRF_Elements.Al_Model[1].B)MOV(CS_XRF.Results[22],CS_XRF_Elements.Al_Scaled);
   52: XIC(CS_XRF.Sts_Running)CPT(CS_XRF.Results[23],CS_XRF_Elements.Al_Model[1].A*CS_XRF_Elements.Al_Model[0].A*XRF_RAWDINT[23]+(CS_XRF_Elements.Al_Model[1].A*CS_XRF_Elements.Al_Model[0].B)+CS_XRF_Elements.Al_Model[1].B)MOV(CS_XRF.Results[23],CS_XRF_Elements.Al_ErrScaled);
   53: XIC(CS_XRF.Sts_Running)CPT(CS_XRF.Results[24],CS_XRF_Elements.Si_Model[1].A*CS_XRF_Elements.Si_Model[0].A*XRF_RAWDINT[24]+(CS_XRF_Elements.Si_Model[1].A*CS_XRF_Elements.Si_Model[0].B)+CS_XRF_Elements.Si_Model[1].B)MOV(CS_XRF.Results[24],CS_XRF_Elements.Si_Scaled);
   54: XIC(CS_XRF.Sts_Running)CPT(CS_XRF.Results[25],CS_XRF_Elements.Si_Model[1].A*CS_XRF_Elements.Si_Model[0].A*XRF_RAWDINT[25]+(CS_XRF_Elements.Si_Model[1].A*CS_XRF_Elements.Si_Model[0].B)+CS_XRF_Elements.Si_Model[1].B)MOV(CS_XRF.Results[25],CS_XRF_Elements.Si_ErrScaled);
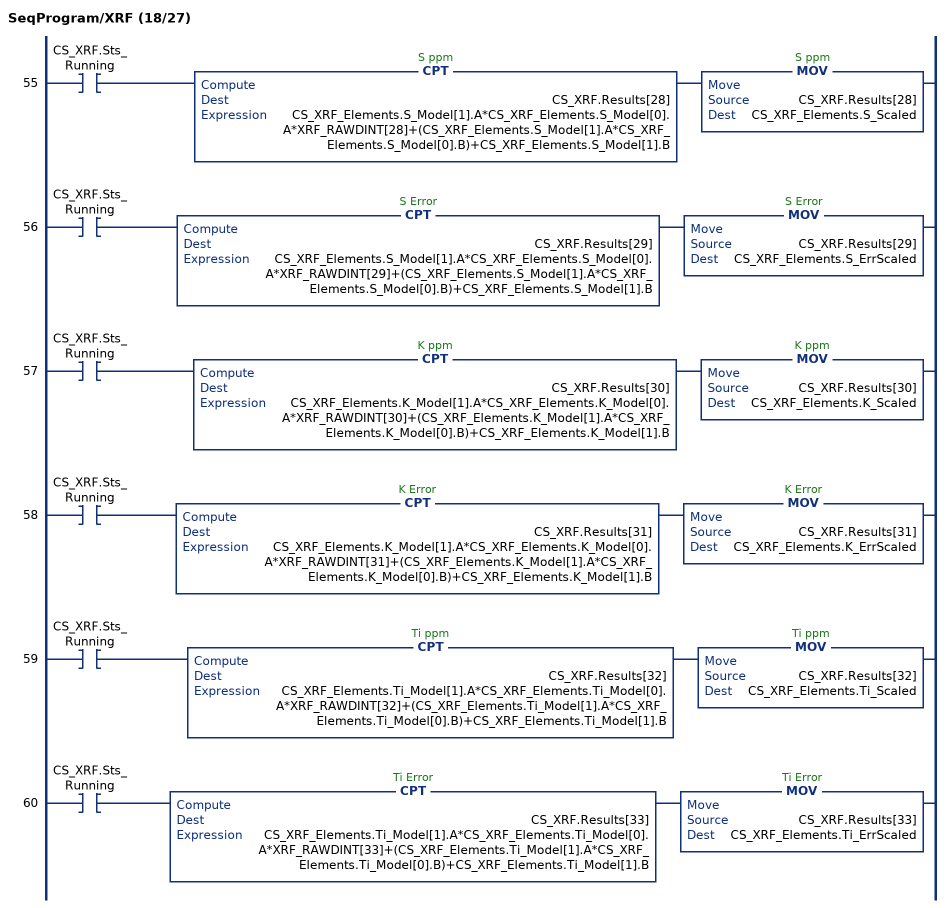
   55: XIC(CS_XRF.Sts_Running)CPT(CS_XRF.Results[28],CS_XRF_Elements.S_Model[1].A*CS_XRF_Elements.S_Model[0].A*XRF_RAWDINT[28]+(CS_XRF_Elements.S_Model[1].A*CS_XRF_Elements.S_Model[0].B)+CS_XRF_Elements.S_Model[1].B)MOV(CS_XRF.Results[28],CS_XRF_Elements.S_Scaled);
   56: XIC(CS_XRF.Sts_Running)CPT(CS_XRF.Results[29],CS_XRF_Elements.S_Model[1].A*CS_XRF_Elements.S_Model[0].A*XRF_RAWDINT[29]+(CS_XRF_Elements.S_Model[1].A*CS_XRF_Elements.S_Model[0].B)+CS_XRF_Elements.S_Model[1].B)MOV(CS_XRF.Results[29],CS_XRF_Elements.S_ErrScaled);
   57: XIC(CS_XRF.Sts_Running)CPT(CS_XRF.Results[30],CS_XRF_Elements.K_Model[1].A*CS_XRF_Elements.K_Model[0].A*XRF_RAWDINT[30]+(CS_XRF_Elements.K_Model[1].A*CS_XRF_Elements.K_Model[0].B)+CS_XRF_Elements.K_Model[1].B)MOV(CS_XRF.Results[30],CS_XRF_Elements.K_Scaled);
   58: XIC(CS_XRF.Sts_Running)CPT(CS_XRF.Results[31],CS_XRF_Elements.K_Model[1].A*CS_XRF_Elements.K_Model[0].A*XRF_RAWDINT[31]+(CS_XRF_Elements.K_Model[1].A*CS_XRF_Elements.K_Model[0].B)+CS_XRF_Elements.K_Model[1].B)MOV(CS_XRF.Results[31],CS_XRF_Elements.K_ErrScaled);
   59: XIC(CS_XRF.Sts_Running)CPT(CS_XRF.Results[32],CS_XRF_Elements.Ti_Model[1].A*CS_XRF_Elements.Ti_Model[0].A*XRF_RAWDINT[32]+(CS_XRF_Elements.Ti_Model[1].A*CS_XRF_Elements.Ti_Model[0].B)+CS_XRF_Elements.Ti_Model[1].B)MOV(CS_XRF.Results[32],CS_XRF_Elements.Ti_Scaled);
   60: XIC(CS_XRF.Sts_Running)CPT(CS_XRF.Results[33],CS_XRF_Elements.Ti_Model[1].A*CS_XRF_Elements.Ti_Model[0].A*XRF_RAWDINT[33]+(CS_XRF_Elements.Ti_Model[1].A*CS_XRF_Elements.Ti_Model[0].B)+CS_XRF_Elements.Ti_Model[1].B)MOV(CS_XRF.Results[33],CS_XRF_Elements.Ti_ErrScaled);
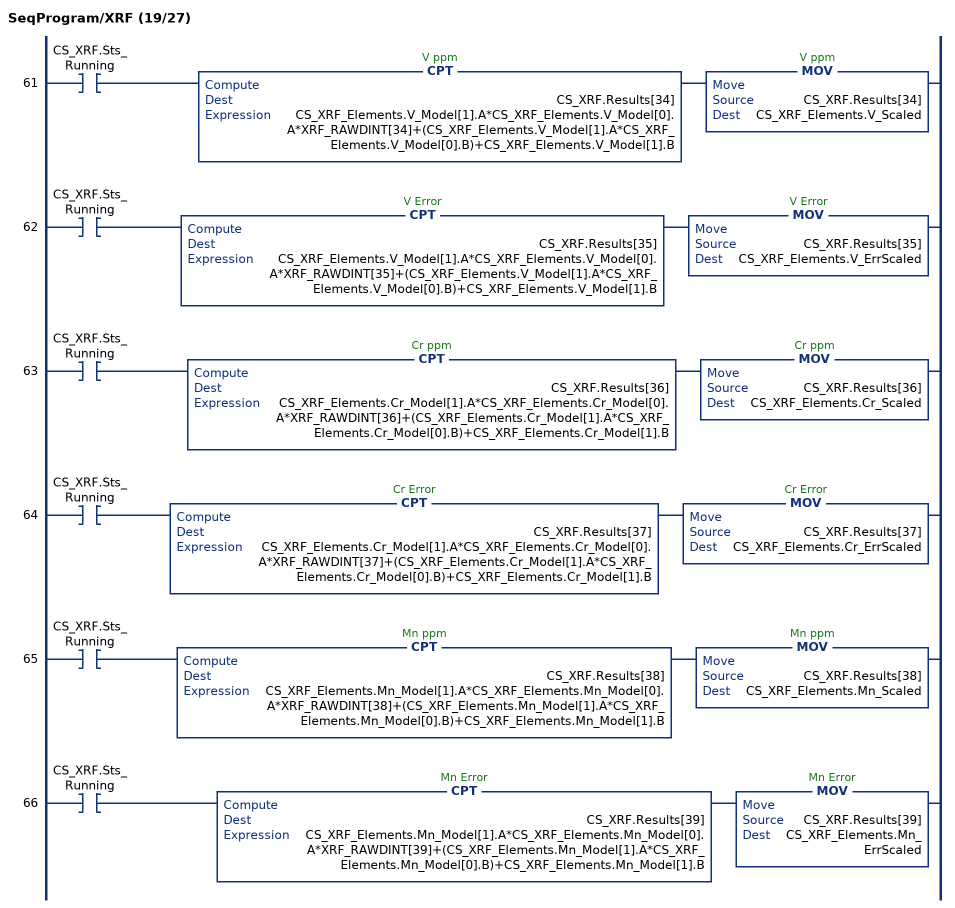
   61: XIC(CS_XRF.Sts_Running)CPT(CS_XRF.Results[34],CS_XRF_Elements.V_Model[1].A*CS_XRF_Elements.V_Model[0].A*XRF_RAWDINT[34]+(CS_XRF_Elements.V_Model[1].A*CS_XRF_Elements.V_Model[0].B)+CS_XRF_Elements.V_Model[1].B)MOV(CS_XRF.Results[34],CS_XRF_Elements.V_Scaled);
   62: XIC(CS_XRF.Sts_Running)CPT(CS_XRF.Results[35],CS_XRF_Elements.V_Model[1].A*CS_XRF_Elements.V_Model[0].A*XRF_RAWDINT[35]+(CS_XRF_Elements.V_Model[1].A*CS_XRF_Elements.V_Model[0].B)+CS_XRF_Elements.V_Model[1].B)MOV(CS_XRF.Results[35],CS_XRF_Elements.V_ErrScaled);
   63: XIC(CS_XRF.Sts_Running)CPT(CS_XRF.Results[36],CS_XRF_Elements.Cr_Model[1].A*CS_XRF_Elements.Cr_Model[0].A*XRF_RAWDINT[36]+(CS_XRF_Elements.Cr_Model[1].A*CS_XRF_Elements.Cr_Model[0].B)+CS_XRF_Elements.Cr_Model[1].B)MOV(CS_XRF.Results[36],CS_XRF_Elements.Cr_Scaled);
   64: XIC(CS_XRF.Sts_Running)CPT(CS_XRF.Results[37],CS_XRF_Elements.Cr_Model[1].A*CS_XRF_Elements.Cr_Model[0].A*XRF_RAWDINT[37]+(CS_XRF_Elements.Cr_Model[1].A*CS_XRF_Elements.Cr_Model[0].B)+CS_XRF_Elements.Cr_Model[1].B)MOV(CS_XRF.Results[37],CS_XRF_Elements.Cr_ErrScaled);
   65: XIC(CS_XRF.Sts_Running)CPT(CS_XRF.Results[38],CS_XRF_Elements.Mn_Model[1].A*CS_XRF_Elements.Mn_Model[0].A*XRF_RAWDINT[38]+(CS_XRF_Elements.Mn_Model[1].A*CS_XRF_Elements.Mn_Model[0].B)+CS_XRF_Elements.Mn_Model[1].B)MOV(CS_XRF.Results[38],CS_XRF_Elements.Mn_Scaled);
   66: XIC(CS_XRF.Sts_Running)CPT(CS_XRF.Results[39],CS_XRF_Elements.Mn_Model[1].A*CS_XRF_Elements.Mn_Model[0].A*XRF_RAWDINT[39]+(CS_XRF_Elements.Mn_Model[1].A*CS_XRF_Elements.Mn_Model[0].B)+CS_XRF_Elements.Mn_Model[1].B)MOV(CS_XRF.Results[39],CS_XRF_Elements.Mn_ErrScaled);
